FUNCTION_BLOCK FB_HMI_VALVES EXTENDS FB_HMI_COMPONENT
VAR_INPUT
END_VAR
VAR_OUTPUT
END_VAR
VAR
END_VAR

END_FUNCTION_BLOCK

(* stored: Version 1.1.0.1, ProductVersion 3.1.4024.14
   POU FB_HMI_VALVES: Id {518a0d1a-2dec-481f-8c88-6d946b728206}, SpecialFunc None *)
